// TIA Portal V17 export
// export: Created 2021-12-03T08:12:57.7155238Z, ExportSetting WithDefaults, DisplayName Totally Integrated Automation Portal, DisplayVersion V17, DisplayName TIA Portal Openness, DisplayVersion V17, DisplayName TIA Portal Version Control Interface, DisplayVersion V17, DisplayName STEP 7 Professional, DisplayVersion V17, DisplayName STEP 7 Safety, DisplayVersion V17, DisplayName WinCC Advanced, DisplayVersion V17
DATA_BLOCK "GDB_Outputs"   // DB90
VERSION : 0.1
// stored: AutoNumber false, IsOnlyStoredInLoadMemory false, IsWriteProtectedInAS false
   VAR RETAIN
      O_PrDoor1Lamp : Bool;   // Protecting Door 1 Lamp
      O_PrDoor2Lamp : Bool;   // Protecting Door 2 Lamp
      O_Spare0_2 : Bool;   // Spare
      O_Spare0_3 : Bool;   // Spare
      O_P3AckInSAreaLamp : Bool;   // Panel 3: Acknowledgement in the Safety Area Lamp
      O_Spare0_5 : Bool;   // Spare
      O_Spare0_6 : Bool;   // Spare
      O_Spare0_7 : Bool;   // Spare
      O_P1AckEmStpOutSAreaLamp : Bool;   // Panel 1: Acknowledgement Emergency Stop outsite the Safety Area Lamp
      O_Spare1_1 : Bool;   // Spare
      O_ChilVlvAcc1 : Bool;   // Accelerator 1 chiller valve
      O_ChilVlvAcc2 : Bool;   // Accelerator 2 chiller valve
      O_P2ConvFwd : Bool;   // Panel 2: Conveyor move forward
      O_P2ConvBwd : Bool;   // Panel 2: Conveyor move backward
      O_ModSwchAcc1 : Bool;   // Accelerator 1 modulator switch
      O_ModSwchAcc2 : Bool;   // Accelerator 2 modulator switch
      O_AccReqWarmUp : Bool;   // Accelerator Request: Warming up
      O_AccReqXRayOn : Bool;   // Accelerator Request: X-Ray on
      O_AccReqXRayNotOn : Bool;   // Accelerator Request: X-Ray not on
      O_AccReqResetFlt : Bool;   // Accelerator Request: Reset Fault
      O_AccReqWarmUpFull : Bool;   // Accelerator Request: Warming up Full (Standby-Clear)
      O_AccReqMicroWaveOn : Bool;   // Accelerator Request: Microwave on
      O_AccReqHighDozeOn : Bool;   // Accelerator Request: HighDoze on
      O_Spare2_7 : Bool;   // Spare
      O_StateSig1RedL : Bool;   // State Signal 1: Red Light
      O_StateSig1YellowL : Bool;   // State Signal 1: Yellow Light
      O_StateSig1GreenL : Bool;   // State Signal 1: Green Light
      O_StateSig1Horn : Bool;   // State Signal 1: Horn
      O_StateSig2WhiteL : Bool;   // State Signal 2: White Light (X-Ray is ON)
      O_Spare3_5 : Bool;   // Spare
      O_Spare3_6 : Bool;   // Spare
      O_StateSig2Horn : Bool;   // State Signal 2: Horn (X-Ray Starts)
   END_VAR
BEGIN
END_DATA_BLOCK
